FUNCTION_BLOCK AngularPosition EXTENDS SM_AngularPosition
VAR_INPUT
END_VAR
VAR_OUTPUT
END_VAR
VAR
    _testVar : INT;
END_VAR

SUPER^();



// do stuff

//SUPER^();

END_FUNCTION_BLOCK

(* stored: Version 1.1.0.1, ProductVersion 3.1.4018.5
   POU AngularPosition: Id {39fd64bb-31c7-4e2a-ba54-df56e455b4a4}, SpecialFunc None *)
